TYPE ST_Horario :
STRUCT
	HoraEntrada : DATE_AND_TIME;
    HoraSalida : DATE_AND_TIME;
END_STRUCT
END_TYPE

(* stored: Version 1.1.0.1, ProductVersion 3.1.4024.12
   DUT ST_Horario: Id {ee93e72c-752a-438b-ba32-482fab7926b6} *)
